FUNCTION_BLOCK WriteOnEdge
VAR_INPUT
	In	: BOOL;
END_VAR

VAR_IN_OUT
	out	:	BOOL;
END_VAR

VAR
	Ftrig	:	f_trig;
	Rtrig	:	r_trig;
END_VAR

//this function block writes the input value to the output, but only when the input changes (falling or rising).
//When no edge detection happens, the output value remains untouched, allowing for parallel input values to 1 output.
//Pair with R_trig on the input for pulse output on input rising edge.

Ftrig(clk := in);
Rtrig(clk := in);

IF (Ftrig.Q OR Rtrig.Q) THEN
	out := in;
END_IF

END_FUNCTION_BLOCK

(* stored: Version 1.1.0.1, ProductVersion 3.1.4026.18
   POU WriteOnEdge: Id {a2aa0500-dd72-49c3-8532-1482c4a69391}, SpecialFunc None *)
